FUNCTION_BLOCK FB_HVFAStorage
VAR_INPUT
END_VAR
VAR_OUTPUT
	UpperTemperature : REAL;
	LowerTemperature : REAL;
END_VAR
VAR
	UpperTemperatureSensor : FB_TemperatureSensor; //upper temperature sensor
	LowerTemperatureSensor : FB_TemperatureSensor; //lower temperature sensor
END_VAR

//get sensor inputs
UpperTemperatureSensor.SetState_AI();
LowerTemperatureSensor.SetState_AI();

//set outputs
UpperTemperature := UpperTemperatureSensor.fTemperature;
LowerTemperature := LowerTemperatureSensor.fTemperature;

END_FUNCTION_BLOCK

(* stored: Version 1.1.0.1, ProductVersion 3.1.4024.10
   POU FB_HVFAStorage: Id {69a5244b-11d5-4395-8b8a-683c8f830970}, SpecialFunc None *)
